// Mitsubishi GX Works2 project: KTFL 20-08-2023_f2   PLC: Q03UDV

PROGRAM MAIN
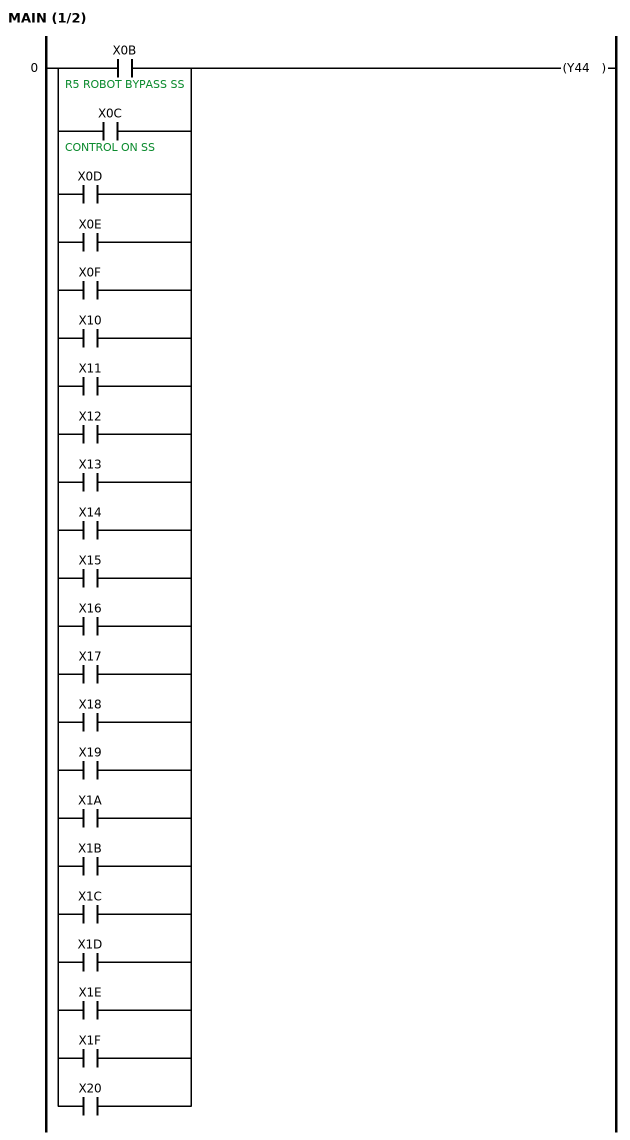
0     LD      X0B  ; R5 ROBOT BYPASS SS
      OR      X0C  ; CONTROL ON SS
      OR      X0D
      OR      X0E
      OR      X0F
      OR      X10
      OR      X11
      OR      X12
      OR      X13
      OR      X14
      OR      X15
      OR      X16
      OR      X17
      OR      X18
      OR      X19
      OR      X1A
      OR      X1B
      OR      X1C
      OR      X1D
      OR      X1E
      OR      X1F
      OR      X20
      OUT     Y44
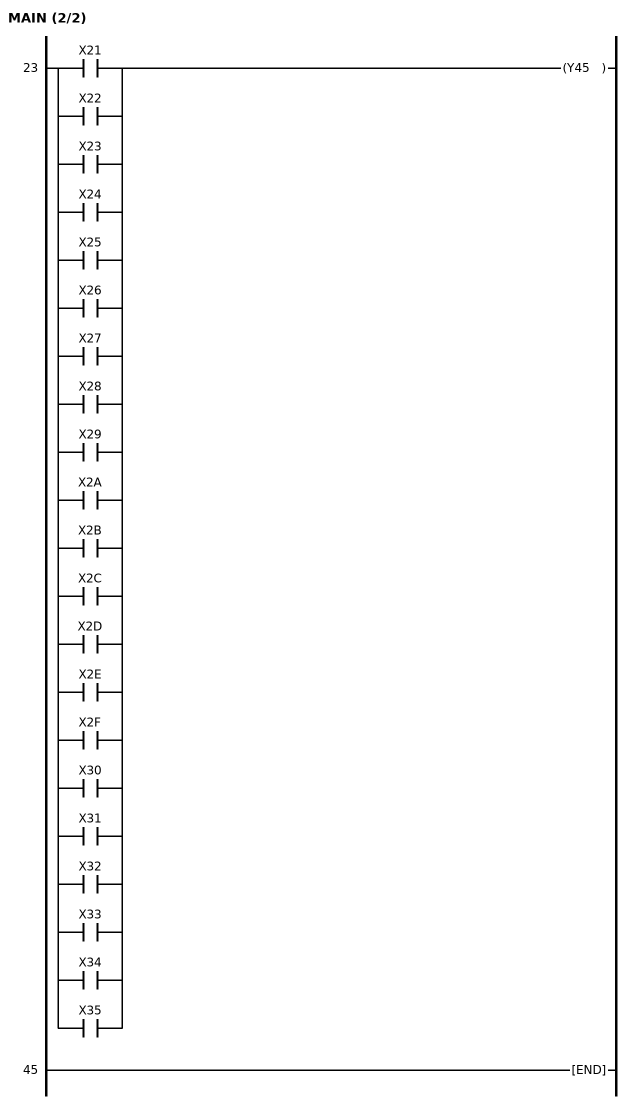
23    LD      X21
      OR      X22
      OR      X23
      OR      X24
      OR      X25
      OR      X26
      OR      X27
      OR      X28
      OR      X29
      OR      X2A
      OR      X2B
      OR      X2C
      OR      X2D
      OR      X2E
      OR      X2F
      OR      X30
      OR      X31
      OR      X32
      OR      X33
      OR      X34
      OR      X35
      OUT     Y45
45    END
END_PROGRAM

PROGRAM DEVICNET
0     END
END_PROGRAM

PROGRAM AUTO_PRG
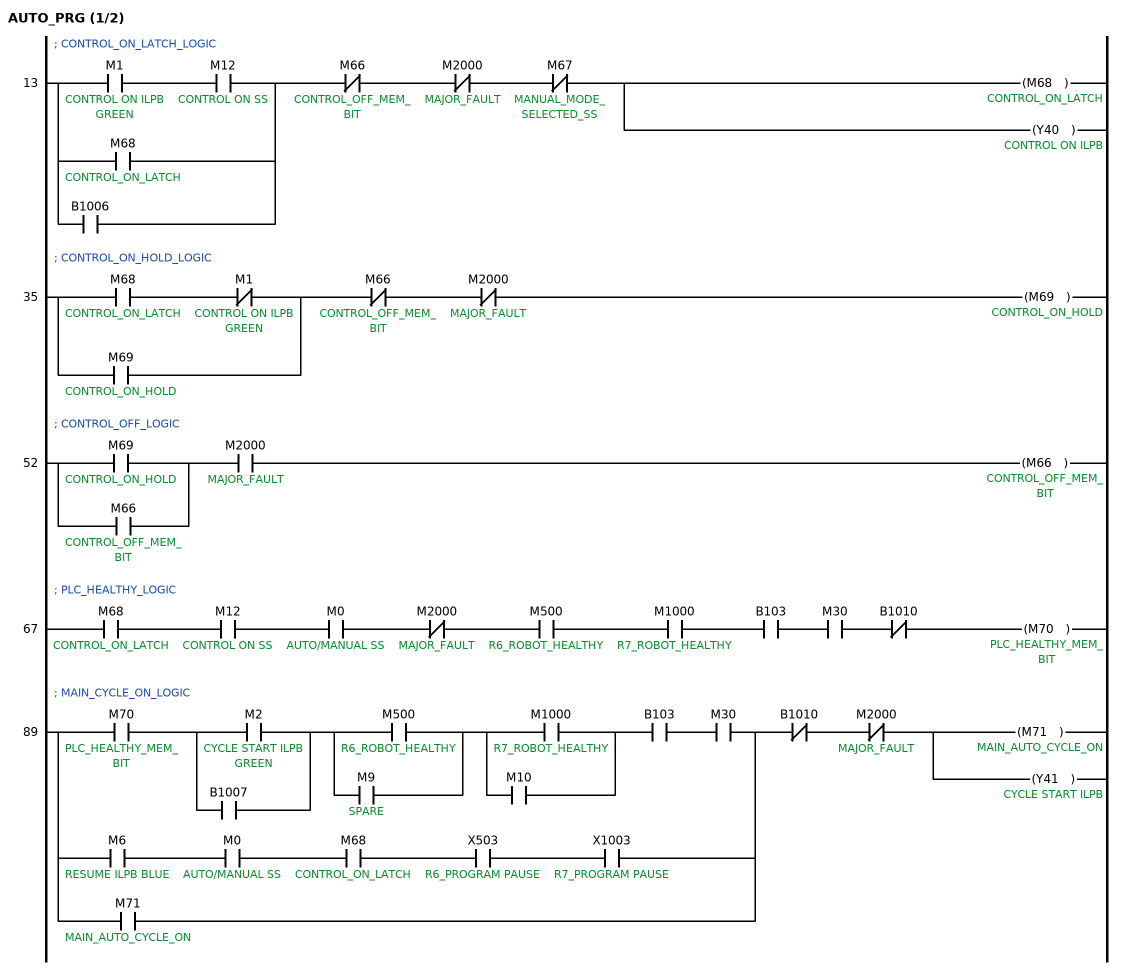
; CONTROL_ON_LATCH_LOGIC
13    LD      M1  ; CONTROL ON ILPB GREEN
      AND     M12  ; CONTROL ON SS
      OR      M68  ; CONTROL_ON_LATCH
      OR      B1006
      ANI     M66  ; CONTROL_OFF_MEM_BIT
      ANI     M2000  ; MAJOR_FAULT
      ANI     M67  ; MANUAL_MODE_SELECTED_SS
      OUT     M68  ; CONTROL_ON_LATCH
      OUT     Y40  ; CONTROL ON ILPB
; CONTROL_ON_HOLD_LOGIC
35    LD      M68  ; CONTROL_ON_LATCH
      ANI     M1  ; CONTROL ON ILPB GREEN
      OR      M69  ; CONTROL_ON_HOLD
      ANI     M66  ; CONTROL_OFF_MEM_BIT
      ANI     M2000  ; MAJOR_FAULT
      OUT     M69  ; CONTROL_ON_HOLD
; CONTROL_OFF_LOGIC
52    LD      M69  ; CONTROL_ON_HOLD
      OR      M66  ; CONTROL_OFF_MEM_BIT
      AND     M2000  ; MAJOR_FAULT
      OUT     M66  ; CONTROL_OFF_MEM_BIT
; PLC_HEALTHY_LOGIC
67    LD      M68  ; CONTROL_ON_LATCH
      AND     M12  ; CONTROL ON SS
      AND     M0  ; AUTO/MANUAL SS
      ANI     M2000  ; MAJOR_FAULT
      AND     M500  ; R6_ROBOT_HEALTHY
      AND     M1000  ; R7_ROBOT_HEALTHY
      AND     B103
      AND     M30
      ANI     B1010
      OUT     M70  ; PLC_HEALTHY_MEM_BIT
; MAIN_CYCLE_ON_LOGIC
89    LD      M70  ; PLC_HEALTHY_MEM_BIT
      LD      M2  ; CYCLE START ILPB GREEN
      OR      B1007
      ANB
      LD      M500  ; R6_ROBOT_HEALTHY
      OR      M9  ; SPARE
      ANB
      LD      M1000  ; R7_ROBOT_HEALTHY
      OR      M10
      ANB
      AND     B103
      AND     M30
      LD      M6  ; RESUME ILPB BLUE
      AND     M0  ; AUTO/MANUAL SS
      AND     M68  ; CONTROL_ON_LATCH
      AND     X503  ; R6_PROGRAM PAUSE
      AND     X1003  ; R7_PROGRAM PAUSE
      ORB
      OR      M71  ; MAIN_AUTO_CYCLE_ON
      ANI     B1010
      ANI     M2000  ; MAJOR_FAULT
      OUT     M71  ; MAIN_AUTO_CYCLE_ON
      OUT     Y41  ; CYCLE START ILPB
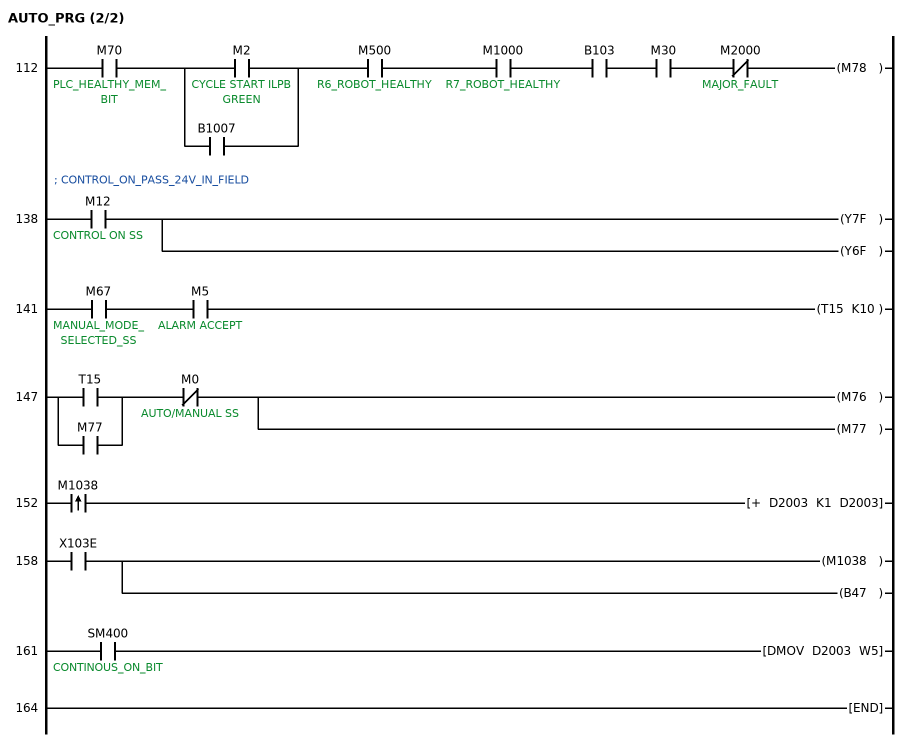
112   LD      M70  ; PLC_HEALTHY_MEM_BIT
      LD      M2  ; CYCLE START ILPB GREEN
      OR      B1007
      ANB
      AND     M500  ; R6_ROBOT_HEALTHY
      AND     M1000  ; R7_ROBOT_HEALTHY
      AND     B103
      AND     M30
      ANI     M2000  ; MAJOR_FAULT
      OUT     M78
; CONTROL_ON_PASS_24V_IN_FIELD
138   LD      M12  ; CONTROL ON SS
      OUT     Y7F
      OUT     Y6F
141   LD      M67  ; MANUAL_MODE_SELECTED_SS
      AND     M5  ; ALARM ACCEPT
      OUT     T15 K10
147   LD      T15
      OR      M77
      ANI     M0  ; AUTO/MANUAL SS
      OUT     M76
      OUT     M77
152   LDP     M1038
      +       D2003 K1 D2003
158   LD      X103E
      OUT     M1038
      OUT     B47
161   LD      SM400  ; CONTINOUS_ON_BIT
      DMOV    D2003 W5
164   END
END_PROGRAM

PROGRAM CC_LINK
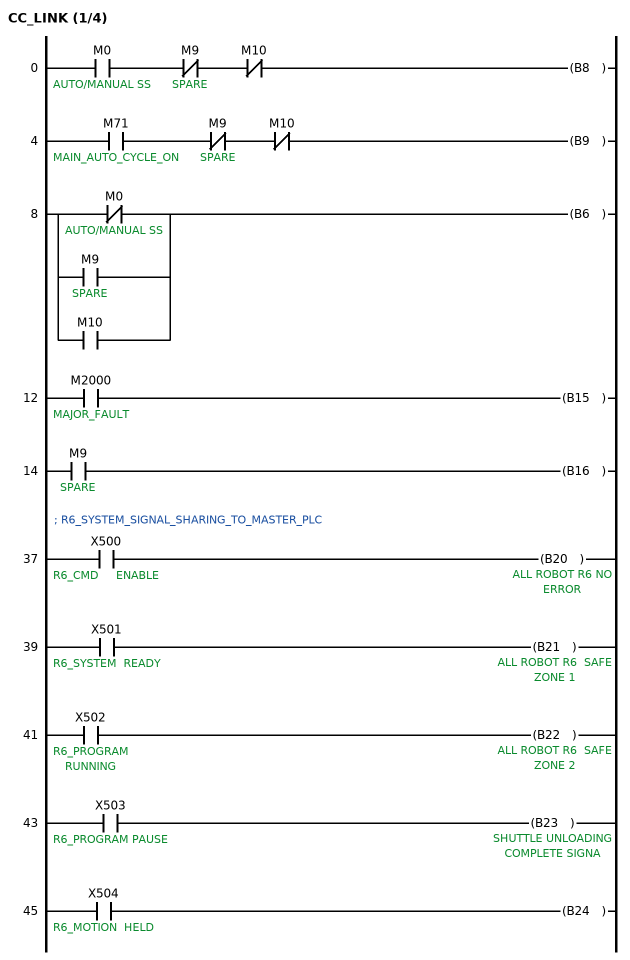
0     LD      M0  ; AUTO/MANUAL SS
      ANI     M9  ; SPARE
      ANI     M10
      OUT     B8
4     LD      M71  ; MAIN_AUTO_CYCLE_ON
      ANI     M9  ; SPARE
      ANI     M10
      OUT     B9
8     LDI     M0  ; AUTO/MANUAL SS
      OR      M9  ; SPARE
      OR      M10
      OUT     B6
12    LD      M2000  ; MAJOR_FAULT
      OUT     B15
14    LD      M9  ; SPARE
      OUT     B16
; R6_SYSTEM_SIGNAL_SHARING_TO_MASTER_PLC
37    LD      X500  ; R6_CMD     ENABLE
      OUT     B20  ; ALL ROBOT R6 NO ERROR
39    LD      X501  ; R6_SYSTEM  READY
      OUT     B21  ; ALL ROBOT R6  SAFE ZONE 1
41    LD      X502  ; R6_PROGRAM RUNNING
      OUT     B22  ; ALL ROBOT R6  SAFE ZONE 2
43    LD      X503  ; R6_PROGRAM PAUSE
      OUT     B23  ; SHUTTLE UNLOADING COMPLETE SIGNA
45    LD      X504  ; R6_MOTION  HELD
      OUT     B24
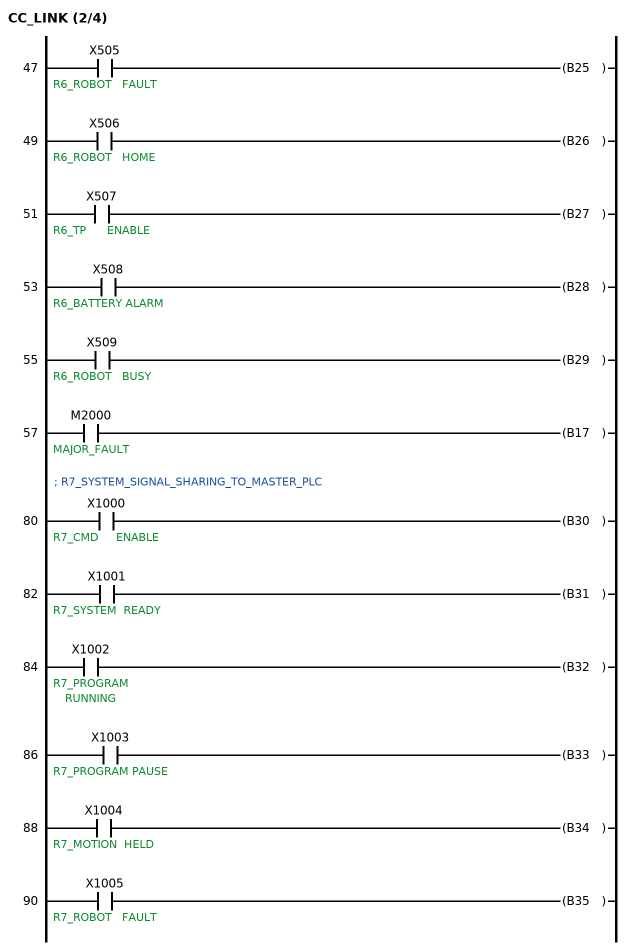
47    LD      X505  ; R6_ROBOT   FAULT
      OUT     B25
49    LD      X506  ; R6_ROBOT   HOME
      OUT     B26
51    LD      X507  ; R6_TP      ENABLE
      OUT     B27
53    LD      X508  ; R6_BATTERY ALARM
      OUT     B28
55    LD      X509  ; R6_ROBOT   BUSY
      OUT     B29
57    LD      M2000  ; MAJOR_FAULT
      OUT     B17
; R7_SYSTEM_SIGNAL_SHARING_TO_MASTER_PLC
80    LD      X1000  ; R7_CMD     ENABLE
      OUT     B30
82    LD      X1001  ; R7_SYSTEM  READY
      OUT     B31
84    LD      X1002  ; R7_PROGRAM RUNNING
      OUT     B32
86    LD      X1003  ; R7_PROGRAM PAUSE
      OUT     B33
88    LD      X1004  ; R7_MOTION  HELD
      OUT     B34
90    LD      X1005  ; R7_ROBOT   FAULT
      OUT     B35
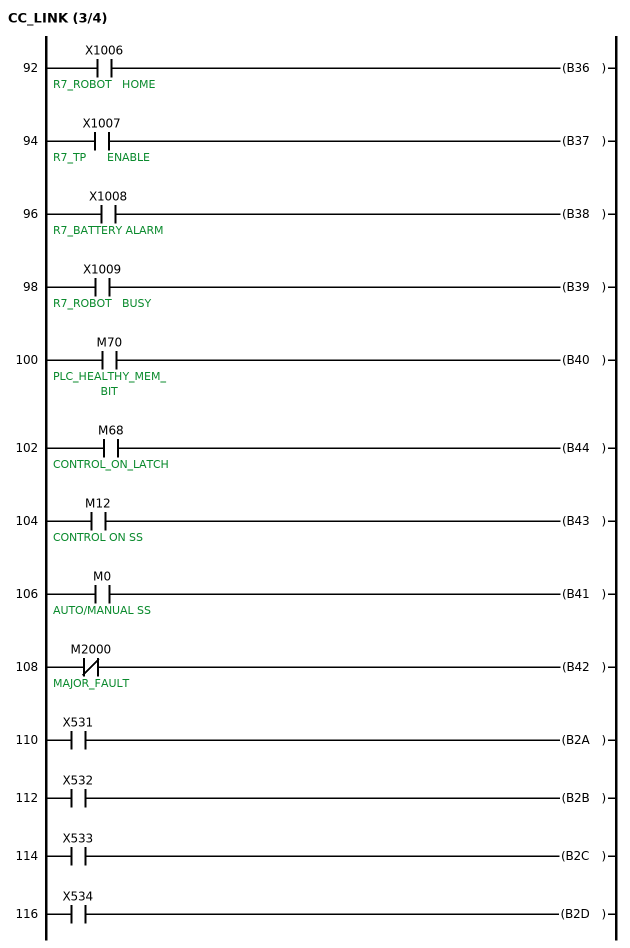
92    LD      X1006  ; R7_ROBOT   HOME
      OUT     B36
94    LD      X1007  ; R7_TP      ENABLE
      OUT     B37
96    LD      X1008  ; R7_BATTERY ALARM
      OUT     B38
98    LD      X1009  ; R7_ROBOT   BUSY
      OUT     B39
100   LD      M70  ; PLC_HEALTHY_MEM_BIT
      OUT     B40
102   LD      M68  ; CONTROL_ON_LATCH
      OUT     B44
104   LD      M12  ; CONTROL ON SS
      OUT     B43
106   LD      M0  ; AUTO/MANUAL SS
      OUT     B41
108   LDI     M2000  ; MAJOR_FAULT
      OUT     B42
110   LD      X531
      OUT     B2A
112   LD      X532
      OUT     B2B
114   LD      X533
      OUT     B2C
116   LD      X534
      OUT     B2D
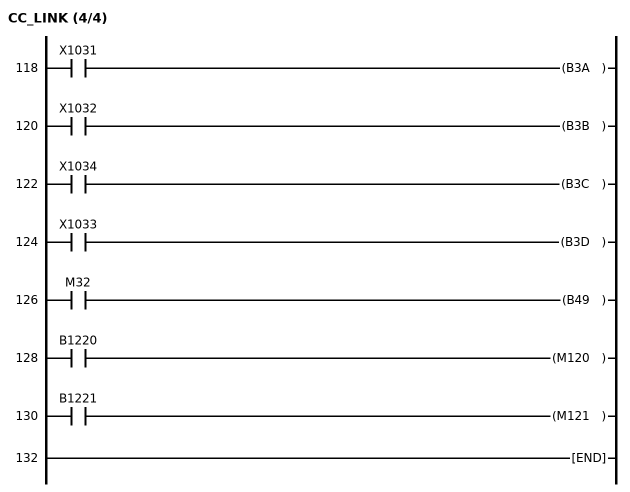
118   LD      X1031
      OUT     B3A
120   LD      X1032
      OUT     B3B
122   LD      X1034
      OUT     B3C
124   LD      X1033
      OUT     B3D
126   LD      M32
      OUT     B49
128   LD      B1220
      OUT     M120
130   LD      B1221
      OUT     M121
132   END
END_PROGRAM

PROGRAM DEVICE_N
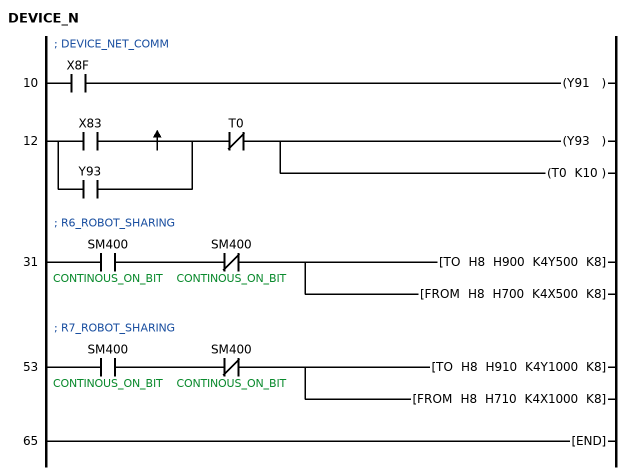
; DEVICE_NET_COMM
10    LD      X8F
      OUT     Y91
12    LD      X83
      MEP
      OR      Y93
      ANI     T0
      OUT     Y93
      OUT     T0 K10
; R6_ROBOT_SHARING
31    LD      SM400  ; CONTINOUS_ON_BIT
      ANI     SM400  ; CONTINOUS_ON_BIT
      TO      H8 H900 K4Y500 K8  ; R6_IMSTP   STOP
      FROM    H8 H700 K4X500 K8  ; R6_CMD     ENABLE
; R7_ROBOT_SHARING
53    LD      SM400  ; CONTINOUS_ON_BIT
      ANI     SM400  ; CONTINOUS_ON_BIT
      TO      H8 H910 K4Y1000 K8  ; R7_IMSTP   STOP
      FROM    H8 H710 K4X1000 K8  ; R7_CMD     ENABLE
65    END
END_PROGRAM

PROGRAM INPUT_MA
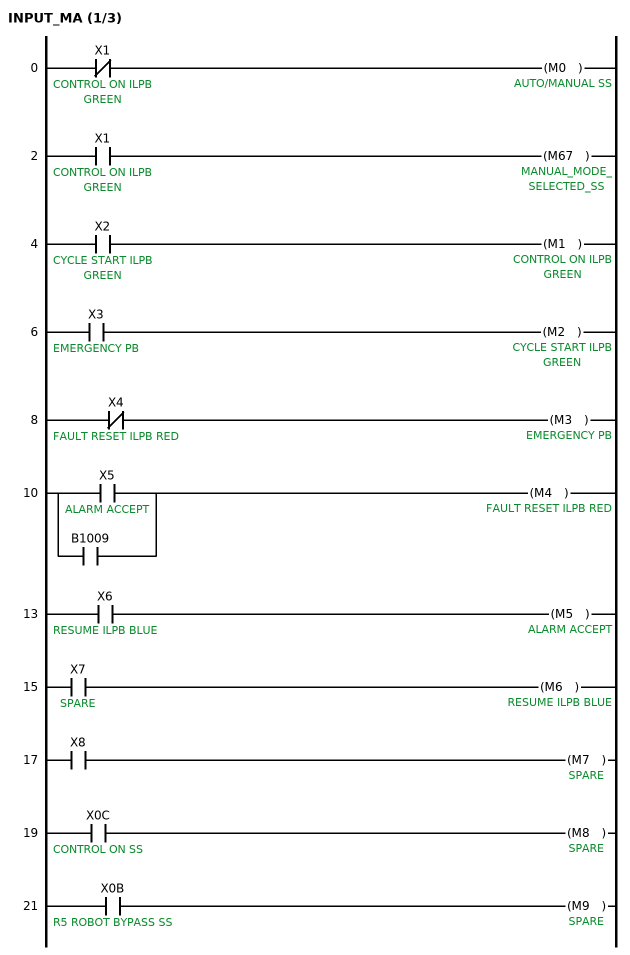
0     LDI     X1  ; CONTROL ON ILPB GREEN
      OUT     M0  ; AUTO/MANUAL SS
2     LD      X1  ; CONTROL ON ILPB GREEN
      OUT     M67  ; MANUAL_MODE_SELECTED_SS
4     LD      X2  ; CYCLE START ILPB GREEN
      OUT     M1  ; CONTROL ON ILPB GREEN
6     LD      X3  ; EMERGENCY PB
      OUT     M2  ; CYCLE START ILPB GREEN
8     LDI     X4  ; FAULT RESET ILPB RED
      OUT     M3  ; EMERGENCY PB
10    LD      X5  ; ALARM ACCEPT
      OR      B1009
      OUT     M4  ; FAULT RESET ILPB RED
13    LD      X6  ; RESUME ILPB BLUE
      OUT     M5  ; ALARM ACCEPT
15    LD      X7  ; SPARE
      OUT     M6  ; RESUME ILPB BLUE
17    LD      X8
      OUT     M7  ; SPARE
19    LD      X0C  ; CONTROL ON SS
      OUT     M8  ; SPARE
21    LD      X0B  ; R5 ROBOT BYPASS SS
      OUT     M9  ; SPARE
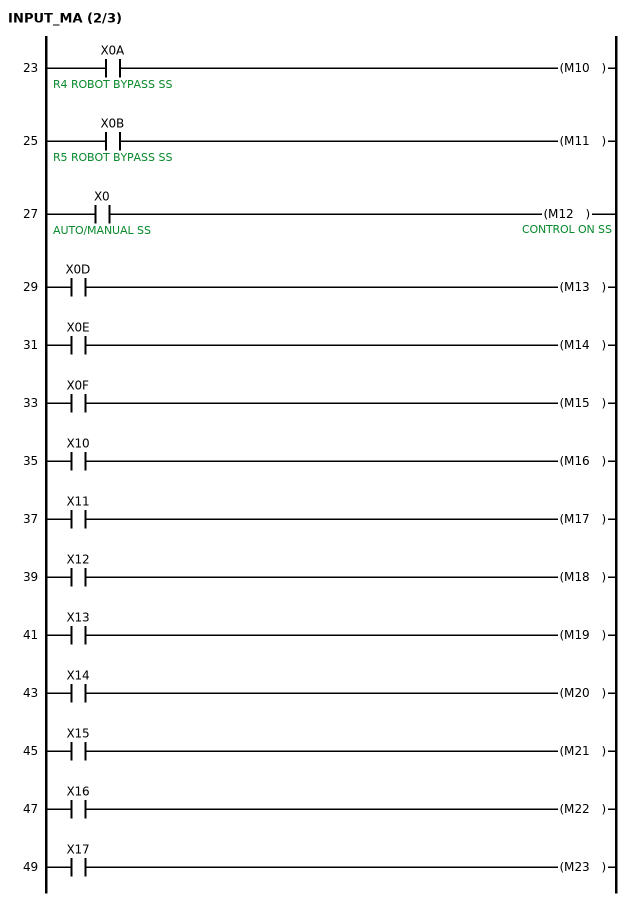
23    LD      X0A  ; R4 ROBOT BYPASS SS
      OUT     M10
25    LD      X0B  ; R5 ROBOT BYPASS SS
      OUT     M11
27    LD      X0  ; AUTO/MANUAL SS
      OUT     M12  ; CONTROL ON SS
29    LD      X0D
      OUT     M13
31    LD      X0E
      OUT     M14
33    LD      X0F
      OUT     M15
35    LD      X10
      OUT     M16
37    LD      X11
      OUT     M17
39    LD      X12
      OUT     M18
41    LD      X13
      OUT     M19
43    LD      X14
      OUT     M20
45    LD      X15
      OUT     M21
47    LD      X16
      OUT     M22
49    LD      X17
      OUT     M23
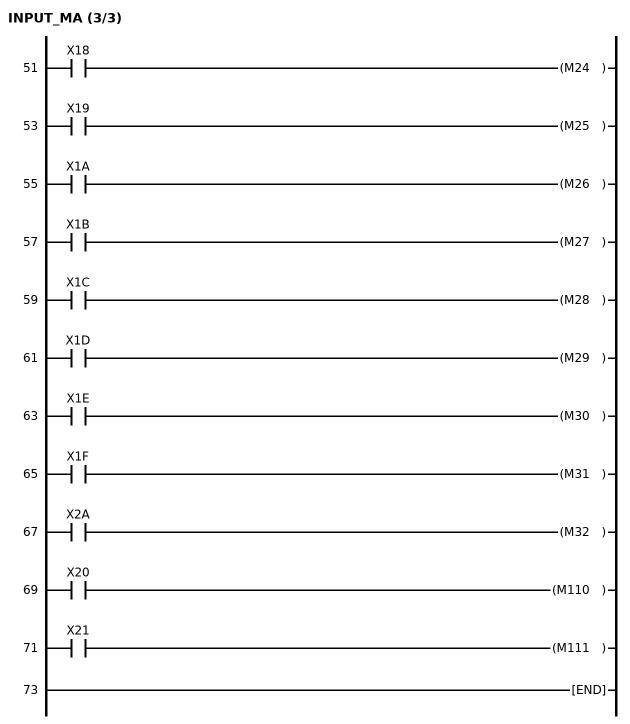
51    LD      X18
      OUT     M24
53    LD      X19
      OUT     M25
55    LD      X1A
      OUT     M26
57    LD      X1B
      OUT     M27
59    LD      X1C
      OUT     M28
61    LD      X1D
      OUT     M29
63    LD      X1E
      OUT     M30
65    LD      X1F
      OUT     M31
67    LD      X2A
      OUT     M32
69    LD      X20
      OUT     M110
71    LD      X21
      OUT     M111
73    END
END_PROGRAM

PROGRAM MANUAL_P
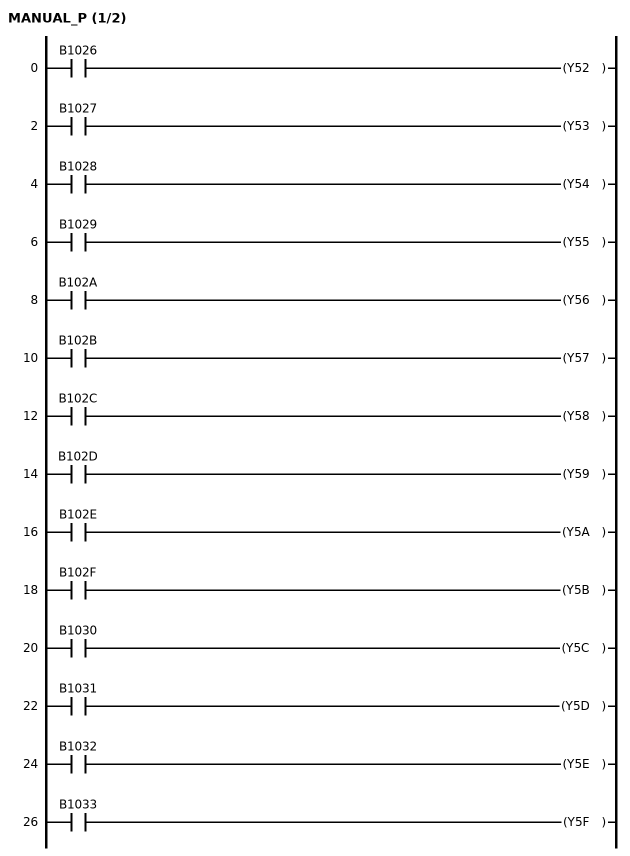
0     LD      B1026
      OUT     Y52
2     LD      B1027
      OUT     Y53
4     LD      B1028
      OUT     Y54
6     LD      B1029
      OUT     Y55
8     LD      B102A
      OUT     Y56
10    LD      B102B
      OUT     Y57
12    LD      B102C
      OUT     Y58
14    LD      B102D
      OUT     Y59
16    LD      B102E
      OUT     Y5A
18    LD      B102F
      OUT     Y5B
20    LD      B1030
      OUT     Y5C
22    LD      B1031
      OUT     Y5D
24    LD      B1032
      OUT     Y5E
26    LD      B1033
      OUT     Y5F
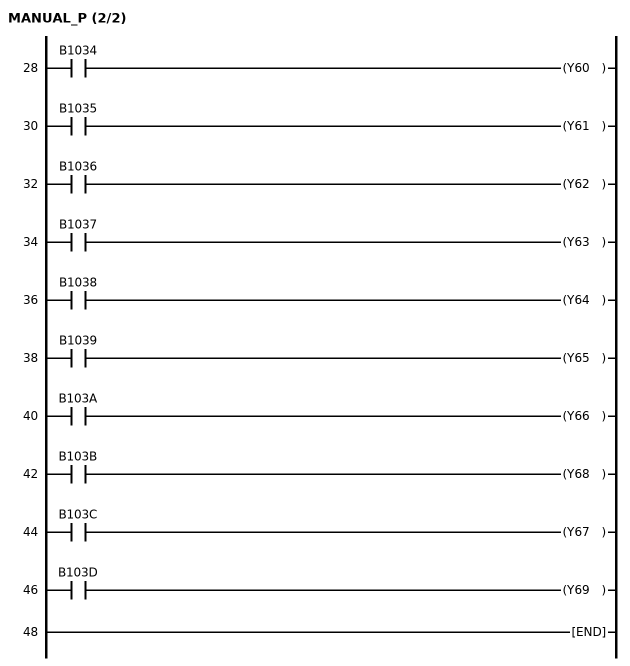
28    LD      B1034
      OUT     Y60
30    LD      B1035
      OUT     Y61
32    LD      B1036
      OUT     Y62
34    LD      B1037
      OUT     Y63
36    LD      B1038
      OUT     Y64
38    LD      B1039
      OUT     Y65
40    LD      B103A
      OUT     Y66
42    LD      B103B
      OUT     Y68
44    LD      B103C
      OUT     Y67
46    LD      B103D
      OUT     Y69
48    END
END_PROGRAM

PROGRAM OUTPUT_M
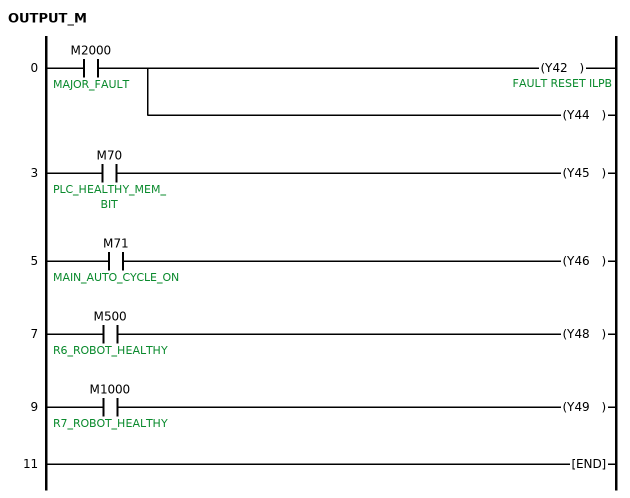
0     LD      M2000  ; MAJOR_FAULT
      OUT     Y42  ; FAULT RESET ILPB
      OUT     Y44
3     LD      M70  ; PLC_HEALTHY_MEM_BIT
      OUT     Y45
5     LD      M71  ; MAIN_AUTO_CYCLE_ON
      OUT     Y46
7     LD      M500  ; R6_ROBOT_HEALTHY
      OUT     Y48
9     LD      M1000  ; R7_ROBOT_HEALTHY
      OUT     Y49
11    END
END_PROGRAM

PROGRAM ROBOT_6
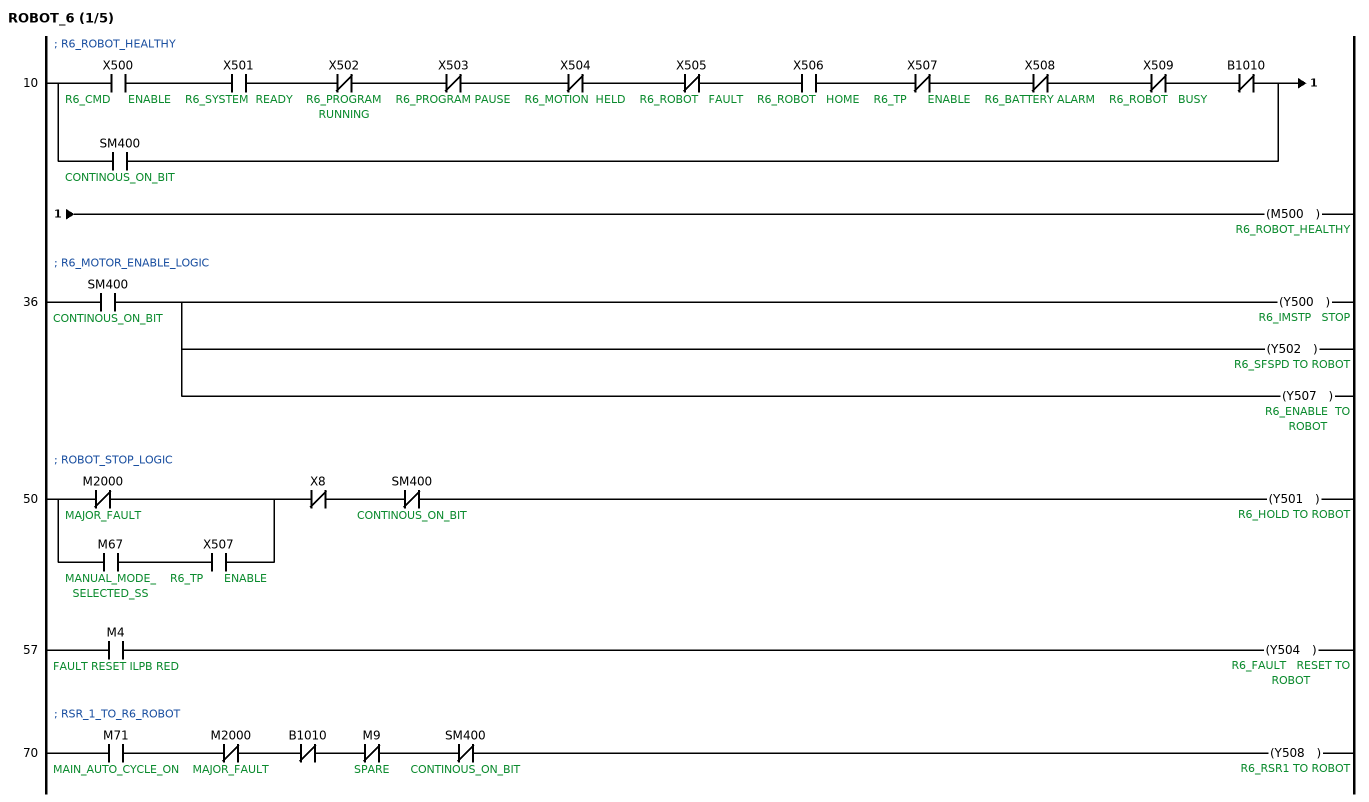
; R6_ROBOT_HEALTHY
10    LD      X500  ; R6_CMD     ENABLE
      AND     X501  ; R6_SYSTEM  READY
      ANI     X502  ; R6_PROGRAM RUNNING
      ANI     X503  ; R6_PROGRAM PAUSE
      ANI     X504  ; R6_MOTION  HELD
      ANI     X505  ; R6_ROBOT   FAULT
      AND     X506  ; R6_ROBOT   HOME
      ANI     X507  ; R6_TP      ENABLE
      ANI     X508  ; R6_BATTERY ALARM
      ANI     X509  ; R6_ROBOT   BUSY
      ANI     B1010
      OR      SM400  ; CONTINOUS_ON_BIT
      OUT     M500  ; R6_ROBOT_HEALTHY
; R6_MOTOR_ENABLE_LOGIC
36    LD      SM400  ; CONTINOUS_ON_BIT
      OUT     Y500  ; R6_IMSTP   STOP
      OUT     Y502  ; R6_SFSPD TO ROBOT
      OUT     Y507  ; R6_ENABLE  TO ROBOT
; ROBOT_STOP_LOGIC
50    LDI     M2000  ; MAJOR_FAULT
      LD      M67  ; MANUAL_MODE_SELECTED_SS
      AND     X507  ; R6_TP      ENABLE
      ORB
      ANI     X8
      ANI     SM400  ; CONTINOUS_ON_BIT
      OUT     Y501  ; R6_HOLD TO ROBOT
57    LD      M4  ; FAULT RESET ILPB RED
      OUT     Y504  ; R6_FAULT   RESET TO ROBOT
; RSR_1_TO_R6_ROBOT
70    LD      M71  ; MAIN_AUTO_CYCLE_ON
      ANI     M2000  ; MAJOR_FAULT
      ANI     B1010
      ANI     M9  ; SPARE
      ANI     SM400  ; CONTINOUS_ON_BIT
      OUT     Y508  ; R6_RSR1 TO ROBOT
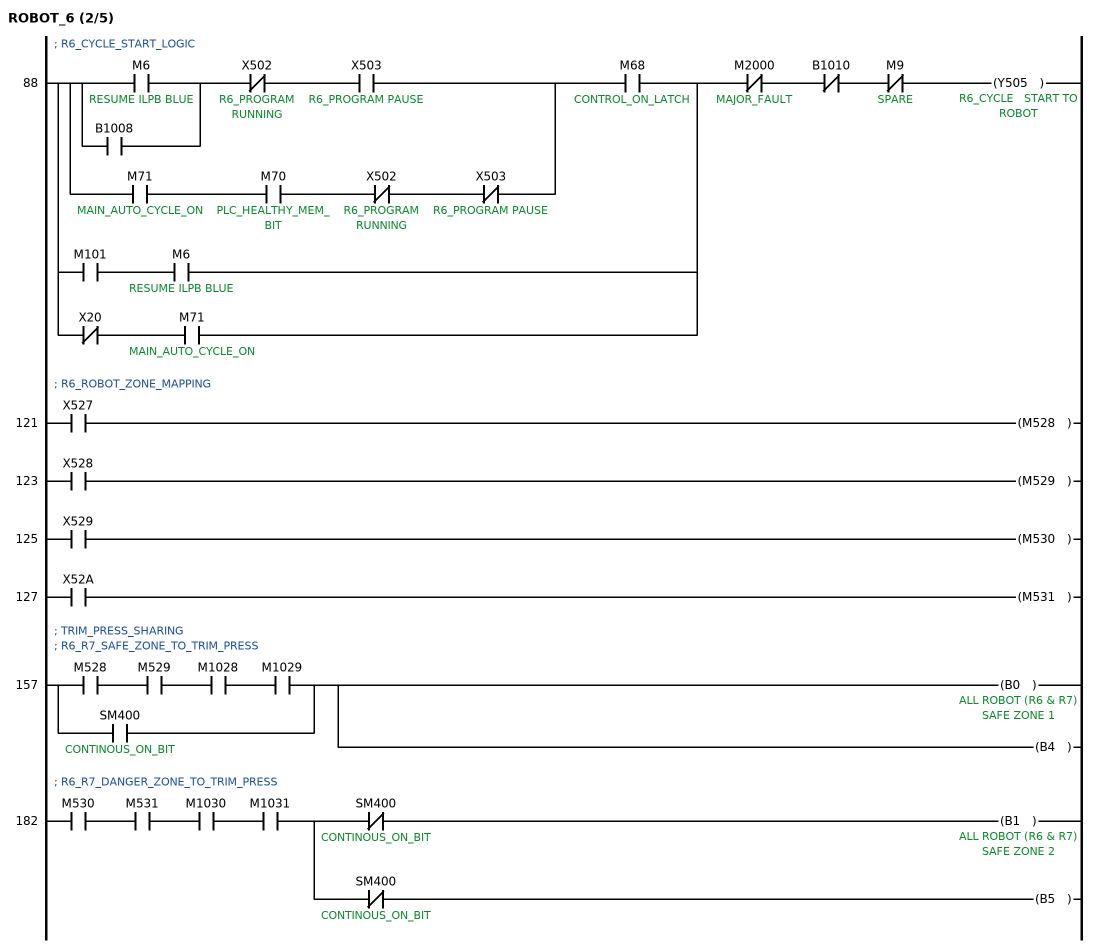
; R6_CYCLE_START_LOGIC
88    LD      M6  ; RESUME ILPB BLUE
      OR      B1008
      ANI     X502  ; R6_PROGRAM RUNNING
      AND     X503  ; R6_PROGRAM PAUSE
      LD      M71  ; MAIN_AUTO_CYCLE_ON
      AND     M70  ; PLC_HEALTHY_MEM_BIT
      ANI     X502  ; R6_PROGRAM RUNNING
      ANI     X503  ; R6_PROGRAM PAUSE
      ORB
      AND     M68  ; CONTROL_ON_LATCH
      LD      M101
      AND     M6  ; RESUME ILPB BLUE
      ORB
      LDI     X20
      AND     M71  ; MAIN_AUTO_CYCLE_ON
      ORB
      ANI     M2000  ; MAJOR_FAULT
      ANI     B1010
      ANI     M9  ; SPARE
      OUT     Y505  ; R6_CYCLE   START TO ROBOT
; R6_ROBOT_ZONE_MAPPING
121   LD      X527
      OUT     M528
123   LD      X528
      OUT     M529
125   LD      X529
      OUT     M530
127   LD      X52A
      OUT     M531
; TRIM_PRESS_SHARING
; R6_R7_SAFE_ZONE_TO_TRIM_PRESS
157   LD      M528
      AND     M529
      AND     M1028
      AND     M1029
      OR      SM400  ; CONTINOUS_ON_BIT
      OUT     B0  ; ALL ROBOT (R6 & R7) SAFE ZONE 1
      OUT     B4
; R6_R7_DANGER_ZONE_TO_TRIM_PRESS
182   LD      M530
      AND     M531
      AND     M1030
      AND     M1031
      MPS
      ANI     SM400  ; CONTINOUS_ON_BIT
      OUT     B1  ; ALL ROBOT (R6 & R7) SAFE ZONE 2
      MPP
      ANI     SM400  ; CONTINOUS_ON_BIT
      OUT     B5
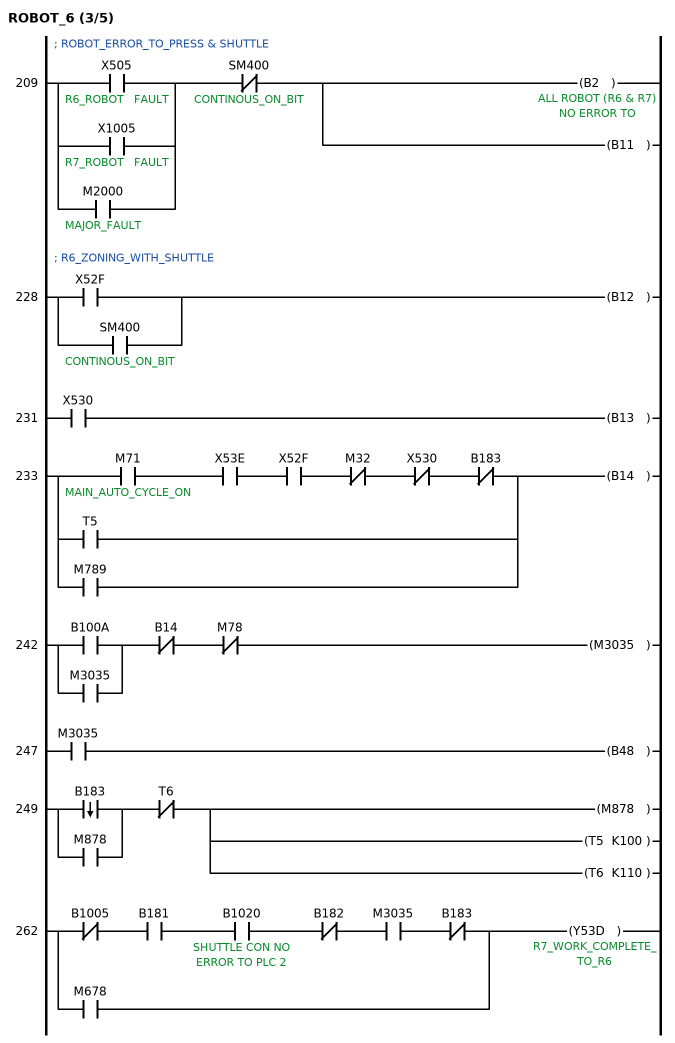
; ROBOT_ERROR_TO_PRESS & SHUTTLE
209   LD      X505  ; R6_ROBOT   FAULT
      OR      X1005  ; R7_ROBOT   FAULT
      OR      M2000  ; MAJOR_FAULT
      ANI     SM400  ; CONTINOUS_ON_BIT
      OUT     B2  ; ALL ROBOT (R6 & R7) NO ERROR TO
      OUT     B11
; R6_ZONING_WITH_SHUTTLE
228   LD      X52F
      OR      SM400  ; CONTINOUS_ON_BIT
      OUT     B12
231   LD      X530
      OUT     B13
233   LD      M71  ; MAIN_AUTO_CYCLE_ON
      AND     X53E
      AND     X52F
      ANI     M32
      ANI     X530
      ANI     B183
      OR      T5
      OR      M789
      OUT     B14
242   LD      B100A
      OR      M3035
      ANI     B14
      ANI     M78
      OUT     M3035
247   LD      M3035
      OUT     B48
249   LDF     B183
      OR      M878
      ANI     T6
      OUT     M878
      OUT     T5 K100
      OUT     T6 K110
262   LDI     B1005
      AND     B181
      AND     B1020  ; SHUTTLE CON NO ERROR TO PLC 2
      ANI     B182
      AND     M3035
      ANI     B183
      OR      M678
      OUT     Y53D  ; R7_WORK_COMPLETE_TO_R6
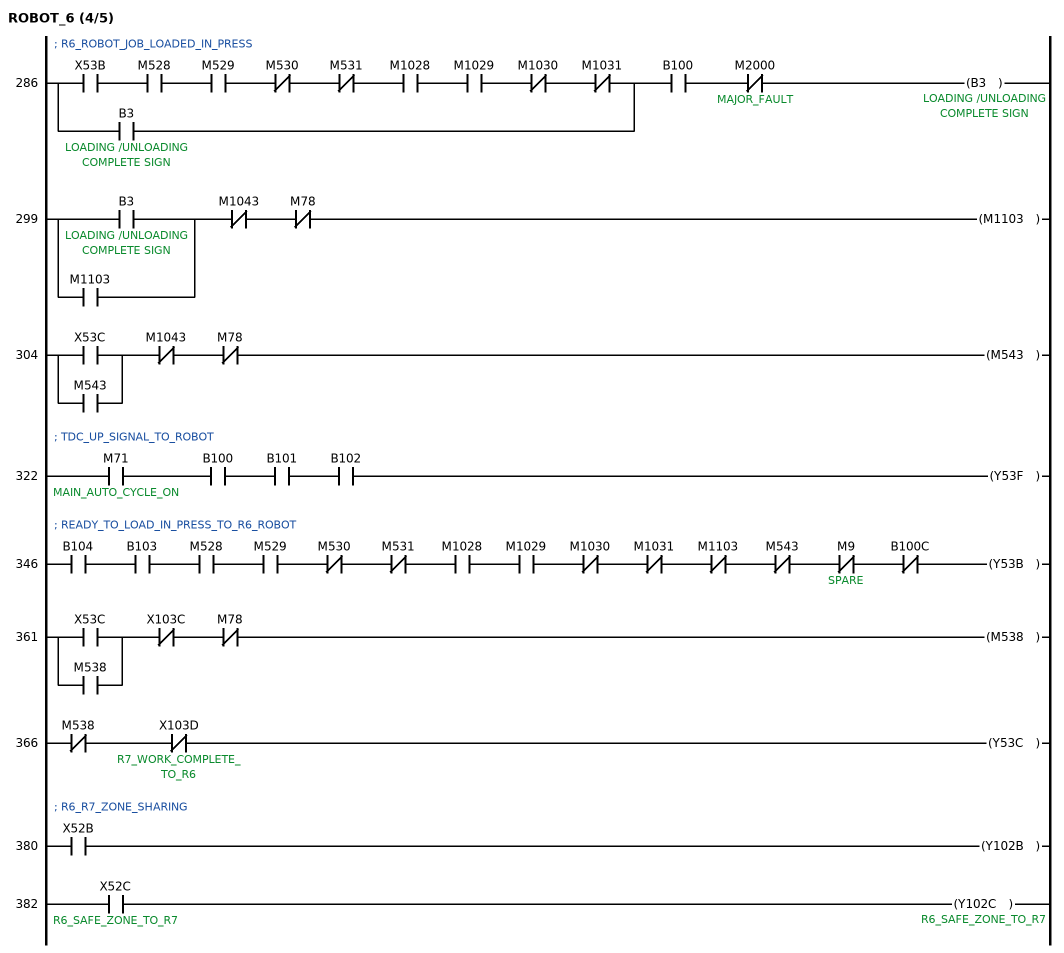
; R6_ROBOT_JOB_LOADED_IN_PRESS
286   LD      X53B
      AND     M528
      AND     M529
      ANI     M530
      ANI     M531
      AND     M1028
      AND     M1029
      ANI     M1030
      ANI     M1031
      OR      B3  ; LOADING /UNLOADING COMPLETE SIGN
      AND     B100
      ANI     M2000  ; MAJOR_FAULT
      OUT     B3  ; LOADING /UNLOADING COMPLETE SIGN
299   LD      B3  ; LOADING /UNLOADING COMPLETE SIGN
      OR      M1103
      ANI     M1043
      ANI     M78
      OUT     M1103
304   LD      X53C
      OR      M543
      ANI     M1043
      ANI     M78
      OUT     M543
; TDC_UP_SIGNAL_TO_ROBOT
322   LD      M71  ; MAIN_AUTO_CYCLE_ON
      AND     B100
      AND     B101
      AND     B102
      OUT     Y53F
; READY_TO_LOAD_IN_PRESS_TO_R6_ROBOT
346   LD      B104
      AND     B103
      AND     M528
      AND     M529
      ANI     M530
      ANI     M531
      AND     M1028
      AND     M1029
      ANI     M1030
      ANI     M1031
      ANI     M1103
      ANI     M543
      ANI     M9  ; SPARE
      ANI     B100C
      OUT     Y53B
361   LD      X53C
      OR      M538
      ANI     X103C
      ANI     M78
      OUT     M538
366   LDI     M538
      ANI     X103D  ; R7_WORK_COMPLETE_TO_R6
      OUT     Y53C
; R6_R7_ZONE_SHARING
380   LD      X52B
      OUT     Y102B
382   LD      X52C  ; R6_SAFE_ZONE_TO_R7
      OUT     Y102C  ; R6_SAFE_ZONE_TO_R7
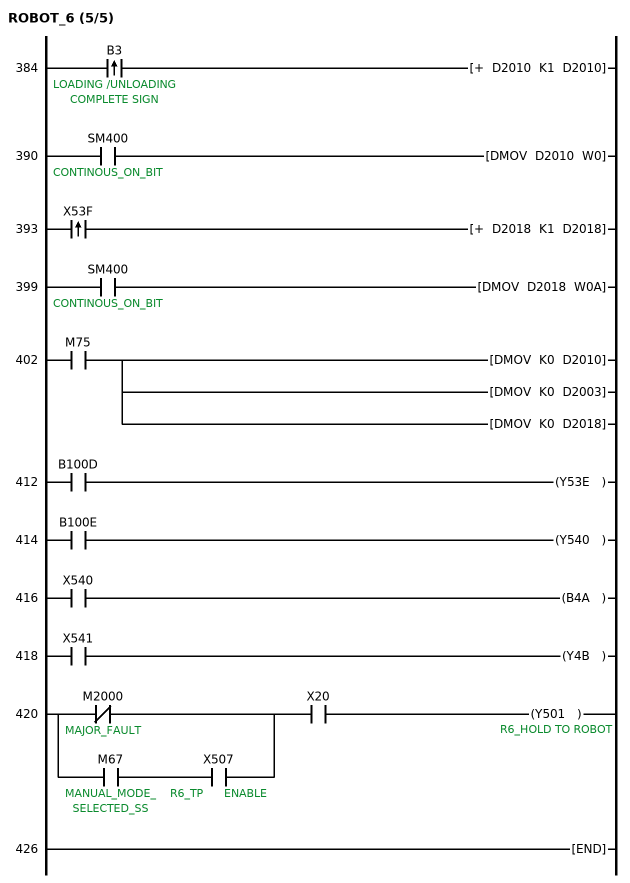
384   LDP     B3  ; LOADING /UNLOADING COMPLETE SIGN
      +       D2010 K1 D2010
390   LD      SM400  ; CONTINOUS_ON_BIT
      DMOV    D2010 W0
393   LDP     X53F
      +       D2018 K1 D2018
399   LD      SM400  ; CONTINOUS_ON_BIT
      DMOV    D2018 W0A
402   LD      M75
      DMOV    K0 D2010
      DMOV    K0 D2003
      DMOV    K0 D2018
412   LD      B100D
      OUT     Y53E
414   LD      B100E
      OUT     Y540
416   LD      X540
      OUT     B4A
418   LD      X541
      OUT     Y4B
420   LDI     M2000  ; MAJOR_FAULT
      LD      M67  ; MANUAL_MODE_SELECTED_SS
      AND     X507  ; R6_TP      ENABLE
      ORB
      AND     X20
      OUT     Y501  ; R6_HOLD TO ROBOT
426   END
END_PROGRAM

PROGRAM ROBOT_7
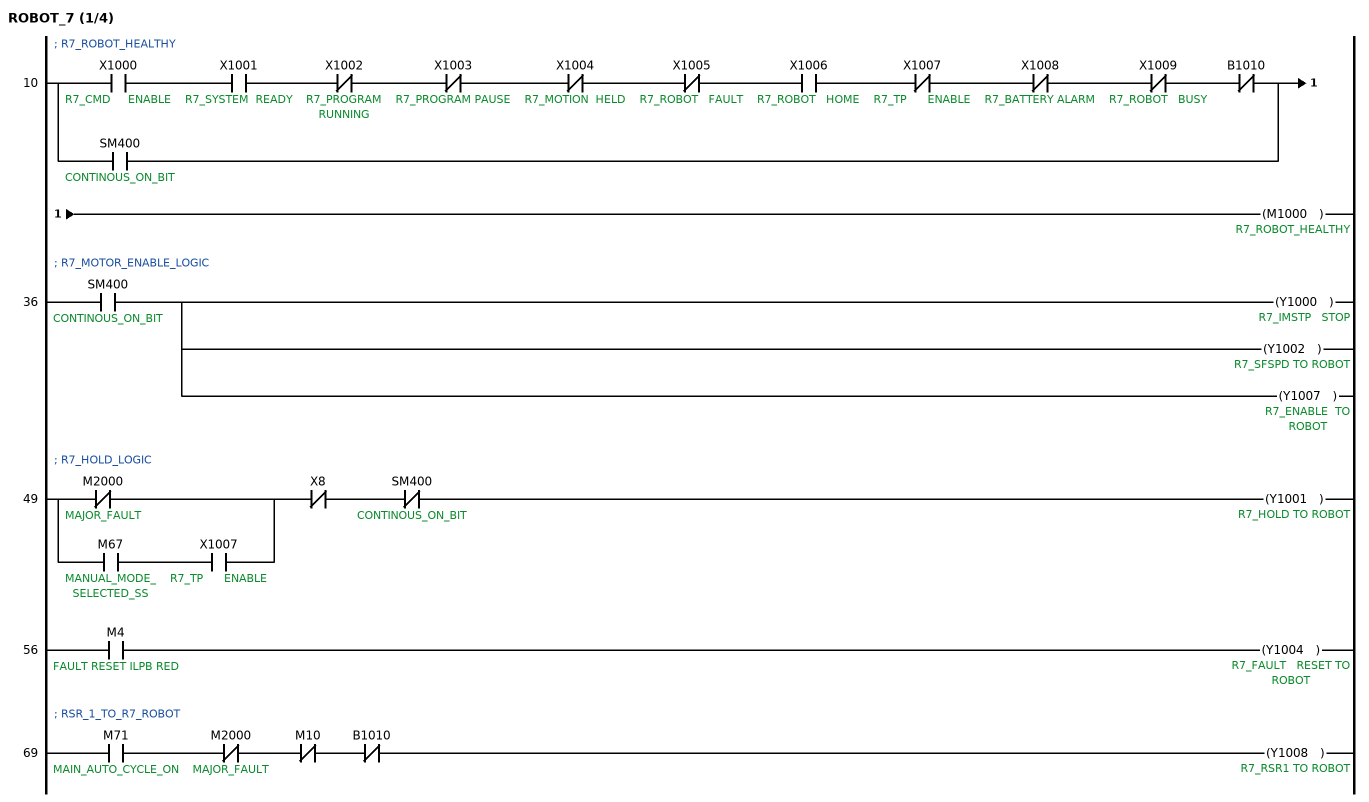
; R7_ROBOT_HEALTHY
10    LD      X1000  ; R7_CMD     ENABLE
      AND     X1001  ; R7_SYSTEM  READY
      ANI     X1002  ; R7_PROGRAM RUNNING
      ANI     X1003  ; R7_PROGRAM PAUSE
      ANI     X1004  ; R7_MOTION  HELD
      ANI     X1005  ; R7_ROBOT   FAULT
      AND     X1006  ; R7_ROBOT   HOME
      ANI     X1007  ; R7_TP      ENABLE
      ANI     X1008  ; R7_BATTERY ALARM
      ANI     X1009  ; R7_ROBOT   BUSY
      ANI     B1010
      OR      SM400  ; CONTINOUS_ON_BIT
      OUT     M1000  ; R7_ROBOT_HEALTHY
; R7_MOTOR_ENABLE_LOGIC
36    LD      SM400  ; CONTINOUS_ON_BIT
      OUT     Y1000  ; R7_IMSTP   STOP
      OUT     Y1002  ; R7_SFSPD TO ROBOT
      OUT     Y1007  ; R7_ENABLE  TO ROBOT
; R7_HOLD_LOGIC
49    LDI     M2000  ; MAJOR_FAULT
      LD      M67  ; MANUAL_MODE_SELECTED_SS
      AND     X1007  ; R7_TP      ENABLE
      ORB
      ANI     X8
      ANI     SM400  ; CONTINOUS_ON_BIT
      OUT     Y1001  ; R7_HOLD TO ROBOT
56    LD      M4  ; FAULT RESET ILPB RED
      OUT     Y1004  ; R7_FAULT   RESET TO ROBOT
; RSR_1_TO_R7_ROBOT
69    LD      M71  ; MAIN_AUTO_CYCLE_ON
      ANI     M2000  ; MAJOR_FAULT
      ANI     M10
      ANI     B1010
      OUT     Y1008  ; R7_RSR1 TO ROBOT
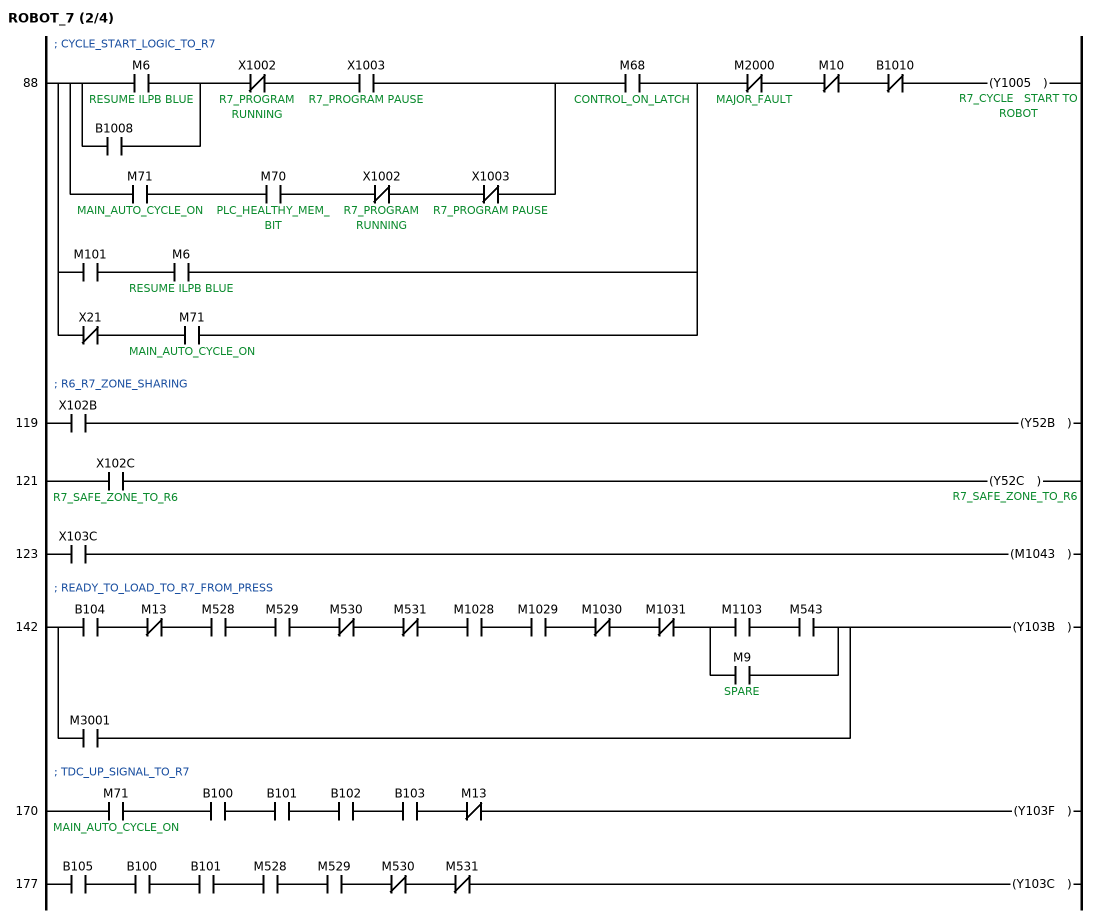
; CYCLE_START_LOGIC_TO_R7
88    LD      M6  ; RESUME ILPB BLUE
      OR      B1008
      ANI     X1002  ; R7_PROGRAM RUNNING
      AND     X1003  ; R7_PROGRAM PAUSE
      LD      M71  ; MAIN_AUTO_CYCLE_ON
      AND     M70  ; PLC_HEALTHY_MEM_BIT
      ANI     X1002  ; R7_PROGRAM RUNNING
      ANI     X1003  ; R7_PROGRAM PAUSE
      ORB
      AND     M68  ; CONTROL_ON_LATCH
      LD      M101
      AND     M6  ; RESUME ILPB BLUE
      ORB
      LDI     X21
      AND     M71  ; MAIN_AUTO_CYCLE_ON
      ORB
      ANI     M2000  ; MAJOR_FAULT
      ANI     M10
      ANI     B1010
      OUT     Y1005  ; R7_CYCLE   START TO ROBOT
; R6_R7_ZONE_SHARING
119   LD      X102B
      OUT     Y52B
121   LD      X102C  ; R7_SAFE_ZONE_TO_R6
      OUT     Y52C  ; R7_SAFE_ZONE_TO_R6
123   LD      X103C
      OUT     M1043
; READY_TO_LOAD_TO_R7_FROM_PRESS
142   LD      B104
      ANI     M13
      AND     M528
      AND     M529
      ANI     M530
      ANI     M531
      AND     M1028
      AND     M1029
      ANI     M1030
      ANI     M1031
      LD      M1103
      AND     M543
      OR      M9  ; SPARE
      ANB
      OR      M3001
      OUT     Y103B
; TDC_UP_SIGNAL_TO_R7
170   LD      M71  ; MAIN_AUTO_CYCLE_ON
      AND     B100
      AND     B101
      AND     B102
      AND     B103
      ANI     M13
      OUT     Y103F
177   LD      B105
      AND     B100
      AND     B101
      AND     M528
      AND     M529
      ANI     M530
      ANI     M531
      OUT     Y103C
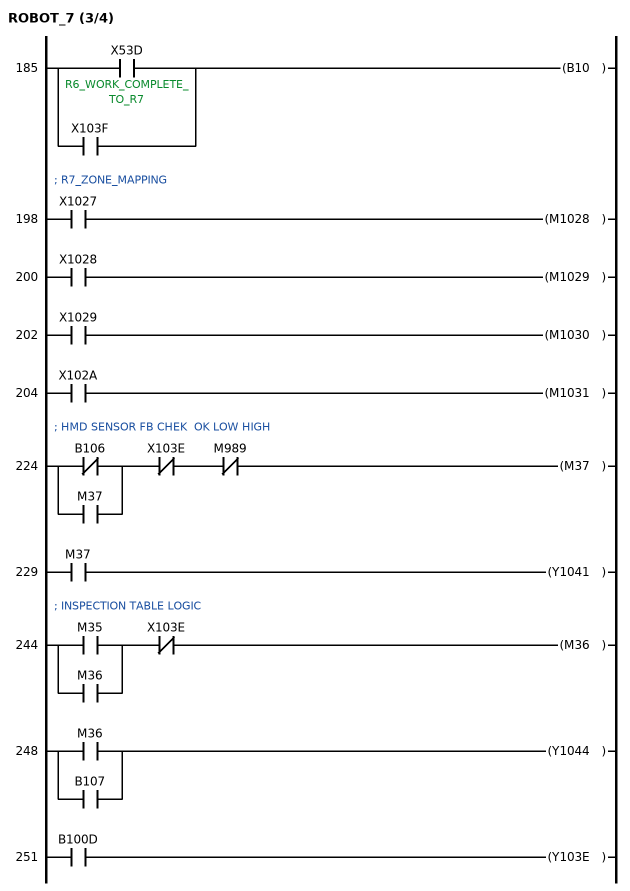
185   LD      X53D  ; R6_WORK_COMPLETE_TO_R7
      OR      X103F
      OUT     B10
; R7_ZONE_MAPPING
198   LD      X1027
      OUT     M1028
200   LD      X1028
      OUT     M1029
202   LD      X1029
      OUT     M1030
204   LD      X102A
      OUT     M1031
; HMD SENSOR FB CHEK  OK LOW HIGH
224   LDI     B106
      OR      M37
      ANI     X103E
      ANI     M989
      OUT     M37
229   LD      M37
      OUT     Y1041
; INSPECTION TABLE LOGIC
244   LD      M35
      OR      M36
      ANI     X103E
      OUT     M36
248   LD      M36
      OR      B107
      OUT     Y1044
251   LD      B100D
      OUT     Y103E
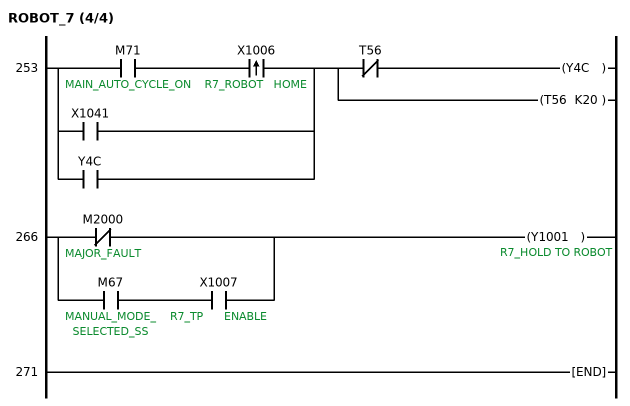
253   LD      M71  ; MAIN_AUTO_CYCLE_ON
      ANDP    X1006  ; R7_ROBOT   HOME
      OR      X1041
      OR      Y4C
      MPS
      ANI     T56
      OUT     Y4C
      MPP
      OUT     T56 K20
266   LDI     M2000  ; MAJOR_FAULT
      LD      M67  ; MANUAL_MODE_SELECTED_SS
      AND     X1007  ; R7_TP      ENABLE
      ORB
      OUT     Y1001  ; R7_HOLD TO ROBOT
271   END
END_PROGRAM

PROGRAM FAULT
